(* CoDeSys 2.3.9.41 project: насос А-М.pro *)
(* Libraries: STANDARD.LIB 4.10.05 11:14:46, IECSFC.LIB 13.4.06 15:51:28, ANALYZATION.LIB 5.10.99 09:05:06 *)

(* PLC configuration (modules and I/O channels)
Discrete input 6 bit [ID100] node 0, in %IB0 out %QB0 {Filtrationtime = 10; Filtrationtime = 10; Filtrationtime = 10; Filtrationtime = 10; Filtrationtime = 10; Filtrationtime = 10; Visibility = Yes; PinCount = 6; WatchDogPeriod = 1000; PollPeriod = 1}
  startPump AT %IX0.0 [BitInput]
  AT %IX0.1 [BitInput]
  AT %IX0.2 [BitInput]
  AT %IX0.3 [BitInput]
  AT %IX0.4 [BitInput]
  AT %IX0.5 [BitInput]
Discrete output 4 bit [ID101] node 1, in %IB1 out %QB1 {PinCount = 4; SafeValueBool = FALSE; SafeValueBool = FALSE; SafeValueBool = FALSE; SafeValueBool = FALSE; Visibility = Yes}
  pumpPin AT %QX1.0 [BitOutput]
  pumpPin1 AT %QX1.1 [BitOutput]
  pumpPin2 AT %QX1.2 [BitOutput]
  errorPin AT %QX1.3 [BitOutput]
Special output [ID104] node 2, in %IB2 out %QB2 {Visibility = No; PinCount = 1}
  AT %QX2.0 [BitOutput] Special output
Unifed signal sensor [ID700] node 3, in %IB3 out %QB3 {Type_of_sensor700 = IT_0_20; measure_interval = 0.8; ainlow = 0; ainhigh = 20; first_cor_point = 0; first_delta = 0; second_cor_point = 0; second_delta = 0; third_cor_point = 0; third_delta = 0; Visibility = No}
  AT %ID3.0 [FloatInput] Value
  AT %IW3.1 [WordInput] Circular time
  Analog Input [ID107] node 0, in %IB3.0 out %QB3.0
Unifed signal sensor [ID700] node 4, in %IB4 out %QB4 {Type_of_sensor700 = IT_0_20; measure_interval = 0.8; ainlow = 0; ainhigh = 20; first_cor_point = 0; first_delta = 0; second_cor_point = 0; second_delta = 0; third_cor_point = 0; third_delta = 0; Visibility = No}
  AT %ID4.0 [FloatInput] Value
  AT %IW4.1 [WordInput] Circular time
  Analog Input [ID107] node 0, in %IB4.0 out %QB4.0
Unifed signal sensor [ID700] node 5, in %IB5 out %QB5 {Type_of_sensor700 = IT_0_20; measure_interval = 0.8; ainlow = 0; ainhigh = 20; first_cor_point = 0; first_delta = 0; second_cor_point = 0; second_delta = 0; third_cor_point = 0; third_delta = 0; Visibility = No}
  AT %ID5.0 [FloatInput] Value
  AT %IW5.1 [WordInput] Circular time
  Analog Input [ID107] node 0, in %IB5.0 out %QB5.0
Unifed signal sensor [ID700] node 6, in %IB6 out %QB6 {Type_of_sensor700 = IT_0_20; measure_interval = 0.8; ainlow = 0; ainhigh = 20; first_cor_point = 0; first_delta = 0; second_cor_point = 0; second_delta = 0; third_cor_point = 0; third_delta = 0; Visibility = Yes}
  AT %ID6.0 [FloatInput] Value
  AT %IW6.1 [WordInput] Circular time
  Analog Input [ID107] node 0, in %IB6.0 out %QB6.0
Analog output [ID106] node 7, in %IB7 out %QB7 {DAC_Type = Voltage 0-10 B; Analog_offset_correction = 0; Analog_full_range_correction = 0; SafeValueFloat = 0; Visibility = No}
  AT %QD7.0 [FloatOutput] Value
Analog output [ID106] node 8, in %IB8 out %QB8 {DAC_Type = Voltage 0-10 B; Analog_offset_correction = 0; Analog_full_range_correction = 0; SafeValueFloat = 0; Visibility = No}
  AT %QD8.0 [FloatOutput] Value
TCP [TCP_ID221] node 0, in %IB9.0.0 out %QB9.0.0 {RemotePort = 502; Visibility = Yes}
PUMP_ON AT %QW9.2.0 [WordOutput]
messag AT %QW9.3.0 [WordOutput]
outGoing AT %QW9.4.0 [WordOutput]
plcStatus AT %QW9.5.0 [WordOutput]
*)

(* POU PLC_PRG, ST *)
PROGRAM PLC_PRG
VAR
	initial:BOOL:=TRUE;
	initTon:TON;
	connectTon:TON;

	PUMP_T:TOF;
	STOP_T:TOF;
	connectCount:INT:=0;
	checkValue:INT:=0;

	(*Параметры для SCADA систем*)
	OPERATOR_PUMP:BOOL:=FALSE;
	OPERATOR_CAN:BOOL:=FALSE;
	OPERATOR_STATUS:INT:=0;

END_VAR
(*Инициализация контроллера*)
IF initial THEN
	pumpPin:=FALSE; pumpPin1:=FALSE;
	pumpPin2:=FALSE; initial:=FALSE;
	initTon.IN:=NOT initial;
END_IF

(*Задержка включения насосов перед отсутствием соединения*)
initTon(PT:=T#20s);
(*Время отсчитываемое до вывода данных об отсутствии сети*)
connectTon(PT:=T#3m);
(*Задержка выключения насоса*)
PUMP_T(PT:=T#10m,);
(*Задержка после нажатия стоп*)
STOP_T(PT:=T#10m,);

(*Проверка подключения системы к другому ПЛК*)
connectTon.IN:=TRUE;
IF plcStatus <> outGoing THEN
	connectTon.IN:=FALSE;
	plcStatus:=outGoing;
	OPERATOR_CAN:=FALSE;
	errorPin:=FALSE;
ELSIF connectTon.Q THEN
	STOP_T.IN:=TRUE;
	OPERATOR_CAN:=TRUE;
	OPERATOR_STATUS:=6;
	PUMP_ON:=0;
	errorPin:=TRUE;
END_IF;


(*Нажата кнопка запуска двигателей*)
IF startPump  AND (PUMP_ON <> 5 OR PUMP_ON=0) THEN
	messag:=2;
	OPERATOR_STATUS:=2;
ELSE
	(*Команда: Насос отключен  *)
	messag:=0;
	IF PUMP_ON=0 AND NOT OPERATOR_CAN  THEN
		OPERATOR_STATUS:=0;
		PUMP_T.IN:=   FALSE;
	(* Команда: Насос включен по показаниям или принудительно*)
	ELSIF PUMP_ON=3 OR PUMP_ON=4  THEN
		OPERATOR_STATUS:=PUMP_ON;
		OPERATOR_PUMP:=FALSE;
		PUMP_T.IN:=TRUE;
	(*Насос включен оператором СКАДЫ системы и не остановлен кнопкой стоп на подъеме №2*)
	ELSIF OPERATOR_PUMP AND OPERATOR_CAN AND  PUMP_ON<>5 THEN
		OPERATOR_STATUS:=1;
		messag:=15;
		PUMP_T.IN:=TRUE;
	(*Иначе отключить Насос*)
	ELSE
		PUMP_T.IN:=FALSE;
	END_IF
END_IF

(*Аварийная остановка*)
IF PUMP_ON=5 THEN
	OPERATOR_STATUS:=PUMP_ON;
	STOP_T.IN:=TRUE;	PUMP_T.IN:=FALSE;
	pumpPin:=FALSE;		pumpPin1:=FALSE;	pumpPin2:=FALSE;
ELSIF startPump THEN
	pumpPin:=TRUE;		pumpPin1:=TRUE;	pumpPin2:=TRUE;
ELSE
	STOP_T.IN:=FALSE;
	pumpPin:=PUMP_T.Q AND NOT STOP_T.Q AND (initTon.Q ) ;
	pumpPin1:=pumpPin;	pumpPin2:=pumpPin;
END_IF
END_PROGRAM
